PROGRAM ClearData
VAR
END_VAR

GVL_DAQ.EXT_CTR.CMDDATACLR			:= FALSE;
GVL_DAQ.DATA_OVERFLOW				:= FALSE;

GVL_DAQ.DATA_INDEX					:= 0;
GVL_DAQ.PASS_INDEX					:= 0;
//GVL_MOTION.RUN_INDEX				:= 1;

GVL_DAQ.CSV_ROW						:= 0;
GVL_DAQ.CSV_PASS_COMPARE			:= 0;


MEMSET(ADR(GVL_DAQ.INDEX_COLLECTOR), 0, SIZEOF(GVL_DAQ.INDEX_COLLECTOR));
MEMSET(ADR(GVL_DAQ.RUNTIME_COLLECTOR), 0, SIZEOF(GVL_DAQ.RUNTIME_COLLECTOR));
MEMSET(ADR(GVL_DAQ.KSM), 0, SIZEOF(GVL_DAQ.KSM));
MEMSET(ADR(GVL_DAQ.TIMESTAMP), 0, SIZEOF(GVL_DAQ.TIMESTAMP));
MEMSET(ADR(GVL_DAQ.MASSA), 0, SIZEOF(GVL_DAQ.MASSA));
MEMSET(ADR(GVL_DAQ.KEYENCE), 0, SIZEOF(GVL_DAQ.KEYENCE));
MEMSET(ADR(GVL_DAQ.X), 0, SIZEOF(GVL_DAQ.X));
MEMSET(ADR(GVL_DAQ.Y), 0, SIZEOF(GVL_DAQ.Y));
MEMSET(ADR(GVL_DAQ.Z), 0, SIZEOF(GVL_DAQ.Z));

END_PROGRAM

(* stored: Version 1.1.0.1, ProductVersion 3.1.4026.12
   POU ClearData: Id {fcbf7d25-d07a-483b-af7c-80e3307b1aca}, SpecialFunc None *)
